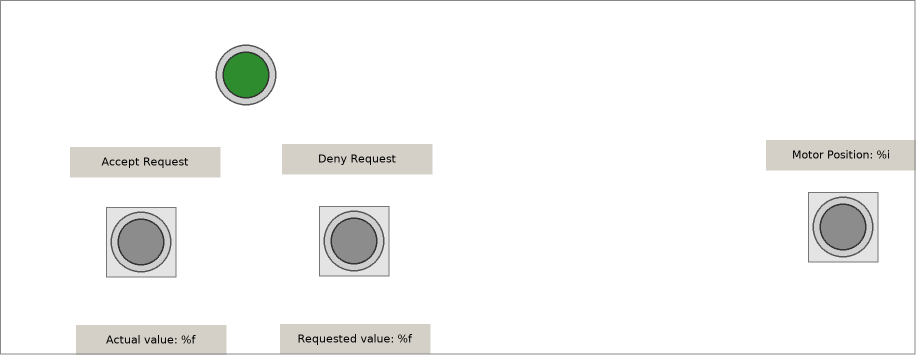
VISUALIZATION Visualization  // 916x355
    PushSwitch (319,206 70x70), variable: MAIN.bDeny, behaviour: TAP, style: Switch-PushSwitch-Gray
    PushSwitch (106,207 70x70), variable: MAIN.bAccept, behaviour: TAP, style: Switch-PushSwitch-Gray
    Textfield (282,144 150x30), "Deny Request"
    Textfield (76,325 150x30), "Actual value: %f", text variable: MAIN.rWrittenValue
    Textfield (70,147 150x30), "Accept Request"
    Textfield (280,324 150x30), "Requested value: %f", text variable: MAIN.rRequestedValue
    Lamp1 (211,40 70x70), variable: MAIN.bRequestIndicator, style: Lamp-Lamp1-Green
    PushSwitch (808,192 70x70), variable: MAIN.bReadPositionButton, behaviour: TAP, style: Switch-PushSwitch-Gray
    Textfield (766,140 150x30), "Motor Position: %i", text variable: MAIN.iPositionMotor
END_VISUALIZATION

(* stored: Version 1.1.0.1, ProductVersion 3.1.4024.5
   Visu Visualization: Id {bcb35772-e08c-488b-9d89-d56a98bcfba1} *)
